FUNCTION remove_project_from_path : STRING(120)
VAR_INPUT
  path: STRING(120);
END_VAR
VAR
  position: INT;
  length: INT;
  i: INT;
  num_dots: INT;
  offset: INT;
END_VAR
VAR CONSTANT
  ASCII_DOT: INT := 46;
END_VAR

WHILE path[i] <> 0 DO
  IF num_dots < 2 THEN
    IF path[i] = ASCII_DOT THEN
      num_dots := num_dots + 1;
    END_IF
  ELSE
    remove_project_from_path[offset] := path[i];
    offset := offset + 1;
	END_IF
  i := i + 1;
END_WHILE
remove_project_from_path[offset] := 0;

END_FUNCTION

(* stored: Version 1.1.0.1, ProductVersion 3.1.4024.9
   POU remove_project_from_path: Id {edc9cf40-9dd4-4a6b-91fb-91c8b6378125}, SpecialFunc None *)
